FUNCTION_BLOCK FB_HwRefTrayLock
VAR_INPUT
	bLock  			AT %Q* : BOOL;
	bUnlock  		AT %Q* : BOOL;
	bDisableHeater 	AT %Q* : BOOL;
END_VAR
VAR_OUTPUT
	bLocked			AT %I* : BOOL;
	bUnlocked		AT %I* : BOOL;
	eCurrentState : E_LockState;
END_VAR
VAR
END_VAR

IF bLocked THEN
	eCurrentState := E_LockState.Locked;
ELSIF bUnlocked THEN
	eCurrentState := E_LockState.Unlocked;
ELSE
	eCurrentState := E_LockState.UNDEFINIED;
END_IF

PROPERTY P_bFeedback : BOOL
GET
P_bFeedback := F_GetMappingStatus(ADR(bLocked), SIZEOF(bLocked)) = EPlcMappingStatus.MS_Partial AND 
				F_GetMappingStatus(ADR(bUnlocked), SIZEOF(bUnlocked)) = EPlcMappingStatus.MS_Partial;
END_GET
END_PROPERTY

END_FUNCTION_BLOCK

(* stored: Version 1.1.0.1
   POU FB_HwRefTrayLock: Id {3eb50bb5-ff53-4ec5-93e8-e5a853092110}, SpecialFunc None
   Property P_bFeedback: Id {c5d9e6ae-98c4-4f67-b4fb-c92036690f22}
   Get Get: Id {10ddd09c-1001-45a2-bc7e-3a657ad3aa4b} *)
